SUBAPPLICATION Uebung_012c_AIS (* String Input und Speichern *)
  (* Standard: 61499-2; Description: Copyright (c) 2023 Meisterschulen am Ostbahnhof This program and the accompanying materials are made available under the terms of the Eclipse Public License 2.0 which is available at https://www.eclipse.org/legal/epl-2.0/ SPDX-License-Identifier: EPL-2.0 *)
  (* Version 1.0, 2026-04-13, Franz Höpfinger, Meisterschulen am Ostbahnhof *)
  PACKAGE Uebungen;
  IMPORT Uebungen::const::NVS::NVS_Keys::KEY_S1_STORE;
  IMPORT Uebungen::const::NVS::NVS_Keys::SECTION_S1_STORE;
  IMPORT Uebungen::const::UT::DefaultPool::InputNumber_I1;
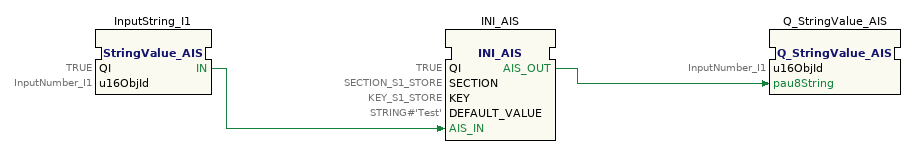
  FBS
    InputString_I1 : isobus::UT::io::StringValue::StringValue_AIS(QI := TRUE, u16ObjId := InputNumber_I1);
    INI_AIS : eclipse4diac::storage::INI_AIS(QI := TRUE, SECTION := SECTION_S1_STORE, KEY := KEY_S1_STORE, DEFAULT_VALUE := STRING#'Test');
    Q_StringValue_AIS : isobus::UT::Q::Q_StringValue_AIS(u16ObjId := InputNumber_I1);
  END_FBS
  ADAPTER_CONNECTIONS
    InputString_I1.IN TO INI_AIS.AIS_IN;
    INI_AIS.AIS_OUT TO Q_StringValue_AIS.pau8String;
  END_CONNECTIONS
END_SUBAPPLICATION
